SUBAPPLICATION InputOutputTesterButton_PWM_OPC_UA (* PWM Tester (OPC-UA): 8 unveraenderte digitale Eingaenge + 12 PWM-Ausgaenge (VT-Zahlenfeld/Balken/6 Ramp-Tasten je Kanal) *)
  (* Standard: 61499-2; Description: Copyright (c) 2026 Meisterschulen am Ostbahnhof This program and the accompanying materials are made available under the terms of the Eclipse Public License 2.0 which is available at https://www.eclipse.org/legal/epl-2.0/ SPDX-License-Identifier: EPL-2.0 *)
  (* Version 1.0, 2026-08-28, Franz Höpfinger, Meisterschulen am Ostbahnhof, initial API and implementation and/or initial documentation *)
  PACKAGE Meins::InputOutputTester::Button_PWM_OPC_UA;
  IMPORT Meins::InputOutputTester::Button_PWM_OPC_UA::SubStrings::I1_WRITE;
  IMPORT Meins::InputOutputTester::Button_PWM_OPC_UA::SubStrings::I2_WRITE;
  IMPORT Meins::InputOutputTester::Button_PWM_OPC_UA::SubStrings::I3_WRITE;
  IMPORT Meins::InputOutputTester::Button_PWM_OPC_UA::SubStrings::I4_WRITE;
  IMPORT Meins::InputOutputTester::Button_PWM_OPC_UA::SubStrings::I5_WRITE;
  IMPORT Meins::InputOutputTester::Button_PWM_OPC_UA::SubStrings::I6_WRITE;
  IMPORT Meins::InputOutputTester::Button_PWM_OPC_UA::SubStrings::I7_WRITE;
  IMPORT Meins::InputOutputTester::Button_PWM_OPC_UA::SubStrings::I8_WRITE;
  IMPORT Meins::InputOutputTester::Button_PWM_OPC_UA::SubStrings::PWM_Q01_READ;
  IMPORT Meins::InputOutputTester::Button_PWM_OPC_UA::SubStrings::PWM_Q01_WRITE;
  IMPORT Meins::InputOutputTester::Button_PWM_OPC_UA::SubStrings::PWM_Q01_SWITCH_READ;
  IMPORT Meins::InputOutputTester::Button_PWM_OPC_UA::SubStrings::PWM_Q01_SWITCH_WRITE;
  IMPORT Meins::InputOutputTester::Button_PWM_OPC_UA::SubStrings::PWM_Q01_STATUS_WRITE;
  IMPORT Meins::InputOutputTester::Button_PWM_OPC_UA::SubStrings::PWM_Q02_READ;
  IMPORT Meins::InputOutputTester::Button_PWM_OPC_UA::SubStrings::PWM_Q02_WRITE;
  IMPORT Meins::InputOutputTester::Button_PWM_OPC_UA::SubStrings::PWM_Q02_SWITCH_READ;
  IMPORT Meins::InputOutputTester::Button_PWM_OPC_UA::SubStrings::PWM_Q02_SWITCH_WRITE;
  IMPORT Meins::InputOutputTester::Button_PWM_OPC_UA::SubStrings::PWM_Q02_STATUS_WRITE;
  IMPORT Meins::InputOutputTester::Button_PWM_OPC_UA::SubStrings::PWM_Q03_READ;
  IMPORT Meins::InputOutputTester::Button_PWM_OPC_UA::SubStrings::PWM_Q03_WRITE;
  IMPORT Meins::InputOutputTester::Button_PWM_OPC_UA::SubStrings::PWM_Q03_SWITCH_READ;
  IMPORT Meins::InputOutputTester::Button_PWM_OPC_UA::SubStrings::PWM_Q03_SWITCH_WRITE;
  IMPORT Meins::InputOutputTester::Button_PWM_OPC_UA::SubStrings::PWM_Q03_STATUS_WRITE;
  IMPORT Meins::InputOutputTester::Button_PWM_OPC_UA::SubStrings::PWM_Q04_READ;
  IMPORT Meins::InputOutputTester::Button_PWM_OPC_UA::SubStrings::PWM_Q04_WRITE;
  IMPORT Meins::InputOutputTester::Button_PWM_OPC_UA::SubStrings::PWM_Q04_SWITCH_READ;
  IMPORT Meins::InputOutputTester::Button_PWM_OPC_UA::SubStrings::PWM_Q04_SWITCH_WRITE;
  IMPORT Meins::InputOutputTester::Button_PWM_OPC_UA::SubStrings::PWM_Q04_STATUS_WRITE;
  IMPORT Meins::InputOutputTester::Button_PWM_OPC_UA::SubStrings::PWM_Q05_READ;
  IMPORT Meins::InputOutputTester::Button_PWM_OPC_UA::SubStrings::PWM_Q05_WRITE;
  IMPORT Meins::InputOutputTester::Button_PWM_OPC_UA::SubStrings::PWM_Q05_SWITCH_READ;
  IMPORT Meins::InputOutputTester::Button_PWM_OPC_UA::SubStrings::PWM_Q05_SWITCH_WRITE;
  IMPORT Meins::InputOutputTester::Button_PWM_OPC_UA::SubStrings::PWM_Q05_STATUS_WRITE;
  IMPORT Meins::InputOutputTester::Button_PWM_OPC_UA::SubStrings::PWM_Q06_READ;
  IMPORT Meins::InputOutputTester::Button_PWM_OPC_UA::SubStrings::PWM_Q06_WRITE;
  IMPORT Meins::InputOutputTester::Button_PWM_OPC_UA::SubStrings::PWM_Q06_SWITCH_READ;
  IMPORT Meins::InputOutputTester::Button_PWM_OPC_UA::SubStrings::PWM_Q06_SWITCH_WRITE;
  IMPORT Meins::InputOutputTester::Button_PWM_OPC_UA::SubStrings::PWM_Q06_STATUS_WRITE;
  IMPORT Meins::InputOutputTester::Button_PWM_OPC_UA::SubStrings::PWM_Q07_READ;
  IMPORT Meins::InputOutputTester::Button_PWM_OPC_UA::SubStrings::PWM_Q07_WRITE;
  IMPORT Meins::InputOutputTester::Button_PWM_OPC_UA::SubStrings::PWM_Q07_SWITCH_READ;
  IMPORT Meins::InputOutputTester::Button_PWM_OPC_UA::SubStrings::PWM_Q07_SWITCH_WRITE;
  IMPORT Meins::InputOutputTester::Button_PWM_OPC_UA::SubStrings::PWM_Q07_STATUS_WRITE;
  IMPORT Meins::InputOutputTester::Button_PWM_OPC_UA::SubStrings::PWM_Q08_READ;
  IMPORT Meins::InputOutputTester::Button_PWM_OPC_UA::SubStrings::PWM_Q08_WRITE;
  IMPORT Meins::InputOutputTester::Button_PWM_OPC_UA::SubStrings::PWM_Q08_SWITCH_READ;
  IMPORT Meins::InputOutputTester::Button_PWM_OPC_UA::SubStrings::PWM_Q08_SWITCH_WRITE;
  IMPORT Meins::InputOutputTester::Button_PWM_OPC_UA::SubStrings::PWM_Q08_STATUS_WRITE;
  IMPORT Meins::InputOutputTester::Button_PWM_OPC_UA::SubStrings::PWM_Q09_READ;
  IMPORT Meins::InputOutputTester::Button_PWM_OPC_UA::SubStrings::PWM_Q09_WRITE;
  IMPORT Meins::InputOutputTester::Button_PWM_OPC_UA::SubStrings::PWM_Q09_SWITCH_READ;
  IMPORT Meins::InputOutputTester::Button_PWM_OPC_UA::SubStrings::PWM_Q09_SWITCH_WRITE;
  IMPORT Meins::InputOutputTester::Button_PWM_OPC_UA::SubStrings::PWM_Q09_STATUS_WRITE;
  IMPORT Meins::InputOutputTester::Button_PWM_OPC_UA::SubStrings::PWM_Q10_READ;
  IMPORT Meins::InputOutputTester::Button_PWM_OPC_UA::SubStrings::PWM_Q10_WRITE;
  IMPORT Meins::InputOutputTester::Button_PWM_OPC_UA::SubStrings::PWM_Q10_SWITCH_READ;
  IMPORT Meins::InputOutputTester::Button_PWM_OPC_UA::SubStrings::PWM_Q10_SWITCH_WRITE;
  IMPORT Meins::InputOutputTester::Button_PWM_OPC_UA::SubStrings::PWM_Q10_STATUS_WRITE;
  IMPORT Meins::InputOutputTester::Button_PWM_OPC_UA::SubStrings::PWM_Q11_READ;
  IMPORT Meins::InputOutputTester::Button_PWM_OPC_UA::SubStrings::PWM_Q11_WRITE;
  IMPORT Meins::InputOutputTester::Button_PWM_OPC_UA::SubStrings::PWM_Q11_SWITCH_READ;
  IMPORT Meins::InputOutputTester::Button_PWM_OPC_UA::SubStrings::PWM_Q11_SWITCH_WRITE;
  IMPORT Meins::InputOutputTester::Button_PWM_OPC_UA::SubStrings::PWM_Q11_STATUS_WRITE;
  IMPORT Meins::InputOutputTester::Button_PWM_OPC_UA::SubStrings::PWM_Q12_READ;
  IMPORT Meins::InputOutputTester::Button_PWM_OPC_UA::SubStrings::PWM_Q12_WRITE;
  IMPORT Meins::InputOutputTester::Button_PWM_OPC_UA::SubStrings::PWM_Q12_SWITCH_READ;
  IMPORT Meins::InputOutputTester::Button_PWM_OPC_UA::SubStrings::PWM_Q12_SWITCH_WRITE;
  IMPORT Meins::InputOutputTester::Button_PWM_OPC_UA::SubStrings::PWM_Q12_STATUS_WRITE;
  IMPORT Meins::InputOutputTester::Button_PWM_OPC_UA::SubStrings::Tick_WRITE;
  IMPORT Uebungen::const::UT::PWM12::DefaultPool_PWM12::Button_I01;
  IMPORT Uebungen::const::UT::PWM12::DefaultPool_PWM12::Button_I02;
  IMPORT Uebungen::const::UT::PWM12::DefaultPool_PWM12::Button_I03;
  IMPORT Uebungen::const::UT::PWM12::DefaultPool_PWM12::Button_I04;
  IMPORT Uebungen::const::UT::PWM12::DefaultPool_PWM12::Button_I05;
  IMPORT Uebungen::const::UT::PWM12::DefaultPool_PWM12::Button_I06;
  IMPORT Uebungen::const::UT::PWM12::DefaultPool_PWM12::Button_I07;
  IMPORT Uebungen::const::UT::PWM12::DefaultPool_PWM12::Button_I08;
  IMPORT Uebungen::const::UT::PWM12::DefaultPool_PWM12::NumberVariable_PWM_Q01;
  IMPORT Uebungen::const::UT::PWM12::DefaultPool_PWM12::Button_PWM_Q01_ZERO;
  IMPORT Uebungen::const::UT::PWM12::DefaultPool_PWM12::Button_PWM_Q01_DOWN_FAST;
  IMPORT Uebungen::const::UT::PWM12::DefaultPool_PWM12::Button_PWM_Q01_DOWN_SLOW;
  IMPORT Uebungen::const::UT::PWM12::DefaultPool_PWM12::Button_PWM_Q01_UP_SLOW;
  IMPORT Uebungen::const::UT::PWM12::DefaultPool_PWM12::Button_PWM_Q01_UP_FAST;
  IMPORT Uebungen::const::UT::PWM12::DefaultPool_PWM12::Button_PWM_Q01_FULL;
  IMPORT Uebungen::const::UT::PWM12::DefaultPool_PWM12::Button_PWM_Q01_SWITCH;
  IMPORT Uebungen::const::UT::PWM12::DefaultPool_PWM12::Button_PWM_Q01_STATUS;
  IMPORT Uebungen::const::UT::PWM12::DefaultPool_PWM12::NumberVariable_PWM_Q02;
  IMPORT Uebungen::const::UT::PWM12::DefaultPool_PWM12::Button_PWM_Q02_ZERO;
  IMPORT Uebungen::const::UT::PWM12::DefaultPool_PWM12::Button_PWM_Q02_DOWN_FAST;
  IMPORT Uebungen::const::UT::PWM12::DefaultPool_PWM12::Button_PWM_Q02_DOWN_SLOW;
  IMPORT Uebungen::const::UT::PWM12::DefaultPool_PWM12::Button_PWM_Q02_UP_SLOW;
  IMPORT Uebungen::const::UT::PWM12::DefaultPool_PWM12::Button_PWM_Q02_UP_FAST;
  IMPORT Uebungen::const::UT::PWM12::DefaultPool_PWM12::Button_PWM_Q02_FULL;
  IMPORT Uebungen::const::UT::PWM12::DefaultPool_PWM12::Button_PWM_Q02_SWITCH;
  IMPORT Uebungen::const::UT::PWM12::DefaultPool_PWM12::Button_PWM_Q02_STATUS;
  IMPORT Uebungen::const::UT::PWM12::DefaultPool_PWM12::NumberVariable_PWM_Q03;
  IMPORT Uebungen::const::UT::PWM12::DefaultPool_PWM12::Button_PWM_Q03_ZERO;
  IMPORT Uebungen::const::UT::PWM12::DefaultPool_PWM12::Button_PWM_Q03_DOWN_FAST;
  IMPORT Uebungen::const::UT::PWM12::DefaultPool_PWM12::Button_PWM_Q03_DOWN_SLOW;
  IMPORT Uebungen::const::UT::PWM12::DefaultPool_PWM12::Button_PWM_Q03_UP_SLOW;
  IMPORT Uebungen::const::UT::PWM12::DefaultPool_PWM12::Button_PWM_Q03_UP_FAST;
  IMPORT Uebungen::const::UT::PWM12::DefaultPool_PWM12::Button_PWM_Q03_FULL;
  IMPORT Uebungen::const::UT::PWM12::DefaultPool_PWM12::Button_PWM_Q03_SWITCH;
  IMPORT Uebungen::const::UT::PWM12::DefaultPool_PWM12::Button_PWM_Q03_STATUS;
  IMPORT Uebungen::const::UT::PWM12::DefaultPool_PWM12::NumberVariable_PWM_Q04;
  IMPORT Uebungen::const::UT::PWM12::DefaultPool_PWM12::Button_PWM_Q04_ZERO;
  IMPORT Uebungen::const::UT::PWM12::DefaultPool_PWM12::Button_PWM_Q04_DOWN_FAST;
  IMPORT Uebungen::const::UT::PWM12::DefaultPool_PWM12::Button_PWM_Q04_DOWN_SLOW;
  IMPORT Uebungen::const::UT::PWM12::DefaultPool_PWM12::Button_PWM_Q04_UP_SLOW;
  IMPORT Uebungen::const::UT::PWM12::DefaultPool_PWM12::Button_PWM_Q04_UP_FAST;
  IMPORT Uebungen::const::UT::PWM12::DefaultPool_PWM12::Button_PWM_Q04_FULL;
  IMPORT Uebungen::const::UT::PWM12::DefaultPool_PWM12::Button_PWM_Q04_SWITCH;
  IMPORT Uebungen::const::UT::PWM12::DefaultPool_PWM12::Button_PWM_Q04_STATUS;
  IMPORT Uebungen::const::UT::PWM12::DefaultPool_PWM12::NumberVariable_PWM_Q05;
  IMPORT Uebungen::const::UT::PWM12::DefaultPool_PWM12::Button_PWM_Q05_ZERO;
  IMPORT Uebungen::const::UT::PWM12::DefaultPool_PWM12::Button_PWM_Q05_DOWN_FAST;
  IMPORT Uebungen::const::UT::PWM12::DefaultPool_PWM12::Button_PWM_Q05_DOWN_SLOW;
  IMPORT Uebungen::const::UT::PWM12::DefaultPool_PWM12::Button_PWM_Q05_UP_SLOW;
  IMPORT Uebungen::const::UT::PWM12::DefaultPool_PWM12::Button_PWM_Q05_UP_FAST;
  IMPORT Uebungen::const::UT::PWM12::DefaultPool_PWM12::Button_PWM_Q05_FULL;
  IMPORT Uebungen::const::UT::PWM12::DefaultPool_PWM12::Button_PWM_Q05_SWITCH;
  IMPORT Uebungen::const::UT::PWM12::DefaultPool_PWM12::Button_PWM_Q05_STATUS;
  IMPORT Uebungen::const::UT::PWM12::DefaultPool_PWM12::NumberVariable_PWM_Q06;
  IMPORT Uebungen::const::UT::PWM12::DefaultPool_PWM12::Button_PWM_Q06_ZERO;
  IMPORT Uebungen::const::UT::PWM12::DefaultPool_PWM12::Button_PWM_Q06_DOWN_FAST;
  IMPORT Uebungen::const::UT::PWM12::DefaultPool_PWM12::Button_PWM_Q06_DOWN_SLOW;
  IMPORT Uebungen::const::UT::PWM12::DefaultPool_PWM12::Button_PWM_Q06_UP_SLOW;
  IMPORT Uebungen::const::UT::PWM12::DefaultPool_PWM12::Button_PWM_Q06_UP_FAST;
  IMPORT Uebungen::const::UT::PWM12::DefaultPool_PWM12::Button_PWM_Q06_FULL;
  IMPORT Uebungen::const::UT::PWM12::DefaultPool_PWM12::Button_PWM_Q06_SWITCH;
  IMPORT Uebungen::const::UT::PWM12::DefaultPool_PWM12::Button_PWM_Q06_STATUS;
  IMPORT Uebungen::const::UT::PWM12::DefaultPool_PWM12::NumberVariable_PWM_Q07;
  IMPORT Uebungen::const::UT::PWM12::DefaultPool_PWM12::Button_PWM_Q07_ZERO;
  IMPORT Uebungen::const::UT::PWM12::DefaultPool_PWM12::Button_PWM_Q07_DOWN_FAST;
  IMPORT Uebungen::const::UT::PWM12::DefaultPool_PWM12::Button_PWM_Q07_DOWN_SLOW;
  IMPORT Uebungen::const::UT::PWM12::DefaultPool_PWM12::Button_PWM_Q07_UP_SLOW;
  IMPORT Uebungen::const::UT::PWM12::DefaultPool_PWM12::Button_PWM_Q07_UP_FAST;
  IMPORT Uebungen::const::UT::PWM12::DefaultPool_PWM12::Button_PWM_Q07_FULL;
  IMPORT Uebungen::const::UT::PWM12::DefaultPool_PWM12::Button_PWM_Q07_SWITCH;
  IMPORT Uebungen::const::UT::PWM12::DefaultPool_PWM12::Button_PWM_Q07_STATUS;
  IMPORT Uebungen::const::UT::PWM12::DefaultPool_PWM12::NumberVariable_PWM_Q08;
  IMPORT Uebungen::const::UT::PWM12::DefaultPool_PWM12::Button_PWM_Q08_ZERO;
  IMPORT Uebungen::const::UT::PWM12::DefaultPool_PWM12::Button_PWM_Q08_DOWN_FAST;
  IMPORT Uebungen::const::UT::PWM12::DefaultPool_PWM12::Button_PWM_Q08_DOWN_SLOW;
  IMPORT Uebungen::const::UT::PWM12::DefaultPool_PWM12::Button_PWM_Q08_UP_SLOW;
  IMPORT Uebungen::const::UT::PWM12::DefaultPool_PWM12::Button_PWM_Q08_UP_FAST;
  IMPORT Uebungen::const::UT::PWM12::DefaultPool_PWM12::Button_PWM_Q08_FULL;
  IMPORT Uebungen::const::UT::PWM12::DefaultPool_PWM12::Button_PWM_Q08_SWITCH;
  IMPORT Uebungen::const::UT::PWM12::DefaultPool_PWM12::Button_PWM_Q08_STATUS;
  IMPORT Uebungen::const::UT::PWM12::DefaultPool_PWM12::NumberVariable_PWM_Q09;
  IMPORT Uebungen::const::UT::PWM12::DefaultPool_PWM12::Button_PWM_Q09_ZERO;
  IMPORT Uebungen::const::UT::PWM12::DefaultPool_PWM12::Button_PWM_Q09_DOWN_FAST;
  IMPORT Uebungen::const::UT::PWM12::DefaultPool_PWM12::Button_PWM_Q09_DOWN_SLOW;
  IMPORT Uebungen::const::UT::PWM12::DefaultPool_PWM12::Button_PWM_Q09_UP_SLOW;
  IMPORT Uebungen::const::UT::PWM12::DefaultPool_PWM12::Button_PWM_Q09_UP_FAST;
  IMPORT Uebungen::const::UT::PWM12::DefaultPool_PWM12::Button_PWM_Q09_FULL;
  IMPORT Uebungen::const::UT::PWM12::DefaultPool_PWM12::Button_PWM_Q09_SWITCH;
  IMPORT Uebungen::const::UT::PWM12::DefaultPool_PWM12::Button_PWM_Q09_STATUS;
  IMPORT Uebungen::const::UT::PWM12::DefaultPool_PWM12::NumberVariable_PWM_Q10;
  IMPORT Uebungen::const::UT::PWM12::DefaultPool_PWM12::Button_PWM_Q10_ZERO;
  IMPORT Uebungen::const::UT::PWM12::DefaultPool_PWM12::Button_PWM_Q10_DOWN_FAST;
  IMPORT Uebungen::const::UT::PWM12::DefaultPool_PWM12::Button_PWM_Q10_DOWN_SLOW;
  IMPORT Uebungen::const::UT::PWM12::DefaultPool_PWM12::Button_PWM_Q10_UP_SLOW;
  IMPORT Uebungen::const::UT::PWM12::DefaultPool_PWM12::Button_PWM_Q10_UP_FAST;
  IMPORT Uebungen::const::UT::PWM12::DefaultPool_PWM12::Button_PWM_Q10_FULL;
  IMPORT Uebungen::const::UT::PWM12::DefaultPool_PWM12::Button_PWM_Q10_SWITCH;
  IMPORT Uebungen::const::UT::PWM12::DefaultPool_PWM12::Button_PWM_Q10_STATUS;
  IMPORT Uebungen::const::UT::PWM12::DefaultPool_PWM12::NumberVariable_PWM_Q11;
  IMPORT Uebungen::const::UT::PWM12::DefaultPool_PWM12::Button_PWM_Q11_ZERO;
  IMPORT Uebungen::const::UT::PWM12::DefaultPool_PWM12::Button_PWM_Q11_DOWN_FAST;
  IMPORT Uebungen::const::UT::PWM12::DefaultPool_PWM12::Button_PWM_Q11_DOWN_SLOW;
  IMPORT Uebungen::const::UT::PWM12::DefaultPool_PWM12::Button_PWM_Q11_UP_SLOW;
  IMPORT Uebungen::const::UT::PWM12::DefaultPool_PWM12::Button_PWM_Q11_UP_FAST;
  IMPORT Uebungen::const::UT::PWM12::DefaultPool_PWM12::Button_PWM_Q11_FULL;
  IMPORT Uebungen::const::UT::PWM12::DefaultPool_PWM12::Button_PWM_Q11_SWITCH;
  IMPORT Uebungen::const::UT::PWM12::DefaultPool_PWM12::Button_PWM_Q11_STATUS;
  IMPORT Uebungen::const::UT::PWM12::DefaultPool_PWM12::NumberVariable_PWM_Q12;
  IMPORT Uebungen::const::UT::PWM12::DefaultPool_PWM12::Button_PWM_Q12_ZERO;
  IMPORT Uebungen::const::UT::PWM12::DefaultPool_PWM12::Button_PWM_Q12_DOWN_FAST;
  IMPORT Uebungen::const::UT::PWM12::DefaultPool_PWM12::Button_PWM_Q12_DOWN_SLOW;
  IMPORT Uebungen::const::UT::PWM12::DefaultPool_PWM12::Button_PWM_Q12_UP_SLOW;
  IMPORT Uebungen::const::UT::PWM12::DefaultPool_PWM12::Button_PWM_Q12_UP_FAST;
  IMPORT Uebungen::const::UT::PWM12::DefaultPool_PWM12::Button_PWM_Q12_FULL;
  IMPORT Uebungen::const::UT::PWM12::DefaultPool_PWM12::Button_PWM_Q12_SWITCH;
  IMPORT Uebungen::const::UT::PWM12::DefaultPool_PWM12::Button_PWM_Q12_STATUS;
  IMPORT Uebungen::const::UT::PWM12::DefaultPool_PWM12::OutputNumber_Tick;
  IMPORT logiBUS::io::DI::logiBUS_DI::Input_I1;
  IMPORT logiBUS::io::DI::logiBUS_DI::Input_I2;
  IMPORT logiBUS::io::DI::logiBUS_DI::Input_I3;
  IMPORT logiBUS::io::DI::logiBUS_DI::Input_I4;
  IMPORT logiBUS::io::DI::logiBUS_DI::Input_I5;
  IMPORT logiBUS::io::DI::logiBUS_DI::Input_I6;
  IMPORT logiBUS::io::DI::logiBUS_DI::Input_I7;
  IMPORT logiBUS::io::DI::logiBUS_DI::Input_I8;
  IMPORT logiBUS::io::DQ::logiBUS_DO::Output_Q1;
  IMPORT logiBUS::io::DQ::logiBUS_DO::Output_Q2;
  IMPORT logiBUS::io::DQ::logiBUS_DO::Output_Q3;
  IMPORT logiBUS::io::DQ::logiBUS_DO::Output_Q4;
  IMPORT logiBUS::io::DQ::logiBUS_DO::Output_Q5;
  IMPORT logiBUS::io::DQ::logiBUS_DO::Output_Q6;
  IMPORT logiBUS::io::DQ::logiBUS_DO::Output_Q7;
  IMPORT logiBUS::io::DQ::logiBUS_DO::Output_Q8;
  IMPORT logiBUS::io::DQ::logiBUS_DO::Output_Q9;
  IMPORT logiBUS::io::DQ::logiBUS_DO::Output_Q10;
  IMPORT logiBUS::io::DQ::logiBUS_DO::Output_Q11;
  IMPORT logiBUS::io::DQ::logiBUS_DO::Output_Q12;
  SUBAPPS
    Input_I1 : MyLib::sys::logiBUS_IXA_BG_OPC(u16ObjId := Button_I01, Input := Input_I1, ID_WRITE := I1_WRITE);
    Input_I2 : MyLib::sys::logiBUS_IXA_BG_OPC(u16ObjId := Button_I02, Input := Input_I2, ID_WRITE := I2_WRITE);
    Input_I3 : MyLib::sys::logiBUS_IXA_BG_OPC(u16ObjId := Button_I03, Input := Input_I3, ID_WRITE := I3_WRITE);
    Input_I4 : MyLib::sys::logiBUS_IXA_BG_OPC(u16ObjId := Button_I04, Input := Input_I4, ID_WRITE := I4_WRITE);
    Input_I5 : MyLib::sys::logiBUS_IXA_BG_OPC(u16ObjId := Button_I05, Input := Input_I5, ID_WRITE := I5_WRITE);
    Input_I6 : MyLib::sys::logiBUS_IXA_BG_OPC(u16ObjId := Button_I06, Input := Input_I6, ID_WRITE := I6_WRITE);
    Input_I7 : MyLib::sys::logiBUS_IXA_BG_OPC(u16ObjId := Button_I07, Input := Input_I7, ID_WRITE := I7_WRITE);
    Input_I8 : MyLib::sys::logiBUS_IXA_BG_OPC(u16ObjId := Button_I08, Input := Input_I8, ID_WRITE := I8_WRITE);
    Output_Q1 : MyLib::sys::RampLimitFS_TO_logiBUS_QDA_PWM_OPC(u16ObjId_VALUEVAR := NumberVariable_PWM_Q01, u16ObjId_SWITCH := Button_PWM_Q01_SWITCH, u16ObjId_STATUS := Button_PWM_Q01_STATUS, bDefaultEnabled := TRUE, u16ObjId_ZERO := Button_PWM_Q01_ZERO, u16ObjId_DOWN_FAST := Button_PWM_Q01_DOWN_FAST, u16ObjId_DOWN_SLOW := Button_PWM_Q01_DOWN_SLOW, u16ObjId_UP_SLOW := Button_PWM_Q01_UP_SLOW, u16ObjId_UP_FAST := Button_PWM_Q01_UP_FAST, u16ObjId_FULL := Button_PWM_Q01_FULL, Output := Output_Q1, ID_READ := PWM_Q01_READ, ID_WRITE := PWM_Q01_WRITE, ID_SWITCH_READ := PWM_Q01_SWITCH_READ, ID_SWITCH_WRITE := PWM_Q01_SWITCH_WRITE, ID_STATUS_WRITE := PWM_Q01_STATUS_WRITE);
    Output_Q2 : MyLib::sys::RampLimitFS_TO_logiBUS_QDA_PWM_OPC(u16ObjId_VALUEVAR := NumberVariable_PWM_Q02, u16ObjId_SWITCH := Button_PWM_Q02_SWITCH, u16ObjId_STATUS := Button_PWM_Q02_STATUS, bDefaultEnabled := TRUE, u16ObjId_ZERO := Button_PWM_Q02_ZERO, u16ObjId_DOWN_FAST := Button_PWM_Q02_DOWN_FAST, u16ObjId_DOWN_SLOW := Button_PWM_Q02_DOWN_SLOW, u16ObjId_UP_SLOW := Button_PWM_Q02_UP_SLOW, u16ObjId_UP_FAST := Button_PWM_Q02_UP_FAST, u16ObjId_FULL := Button_PWM_Q02_FULL, Output := Output_Q2, ID_READ := PWM_Q02_READ, ID_WRITE := PWM_Q02_WRITE, ID_SWITCH_READ := PWM_Q02_SWITCH_READ, ID_SWITCH_WRITE := PWM_Q02_SWITCH_WRITE, ID_STATUS_WRITE := PWM_Q02_STATUS_WRITE);
    Output_Q3 : MyLib::sys::RampLimitFS_TO_logiBUS_QDA_PWM_OPC(u16ObjId_VALUEVAR := NumberVariable_PWM_Q03, u16ObjId_SWITCH := Button_PWM_Q03_SWITCH, u16ObjId_STATUS := Button_PWM_Q03_STATUS, bDefaultEnabled := TRUE, u16ObjId_ZERO := Button_PWM_Q03_ZERO, u16ObjId_DOWN_FAST := Button_PWM_Q03_DOWN_FAST, u16ObjId_DOWN_SLOW := Button_PWM_Q03_DOWN_SLOW, u16ObjId_UP_SLOW := Button_PWM_Q03_UP_SLOW, u16ObjId_UP_FAST := Button_PWM_Q03_UP_FAST, u16ObjId_FULL := Button_PWM_Q03_FULL, Output := Output_Q3, ID_READ := PWM_Q03_READ, ID_WRITE := PWM_Q03_WRITE, ID_SWITCH_READ := PWM_Q03_SWITCH_READ, ID_SWITCH_WRITE := PWM_Q03_SWITCH_WRITE, ID_STATUS_WRITE := PWM_Q03_STATUS_WRITE);
    Output_Q4 : MyLib::sys::RampLimitFS_TO_logiBUS_QDA_PWM_OPC(u16ObjId_VALUEVAR := NumberVariable_PWM_Q04, u16ObjId_SWITCH := Button_PWM_Q04_SWITCH, u16ObjId_STATUS := Button_PWM_Q04_STATUS, bDefaultEnabled := TRUE, u16ObjId_ZERO := Button_PWM_Q04_ZERO, u16ObjId_DOWN_FAST := Button_PWM_Q04_DOWN_FAST, u16ObjId_DOWN_SLOW := Button_PWM_Q04_DOWN_SLOW, u16ObjId_UP_SLOW := Button_PWM_Q04_UP_SLOW, u16ObjId_UP_FAST := Button_PWM_Q04_UP_FAST, u16ObjId_FULL := Button_PWM_Q04_FULL, Output := Output_Q4, ID_READ := PWM_Q04_READ, ID_WRITE := PWM_Q04_WRITE, ID_SWITCH_READ := PWM_Q04_SWITCH_READ, ID_SWITCH_WRITE := PWM_Q04_SWITCH_WRITE, ID_STATUS_WRITE := PWM_Q04_STATUS_WRITE);
    Output_Q5 : MyLib::sys::RampLimitFS_TO_logiBUS_QDA_PWM_OPC(u16ObjId_VALUEVAR := NumberVariable_PWM_Q05, u16ObjId_SWITCH := Button_PWM_Q05_SWITCH, u16ObjId_STATUS := Button_PWM_Q05_STATUS, bDefaultEnabled := TRUE, u16ObjId_ZERO := Button_PWM_Q05_ZERO, u16ObjId_DOWN_FAST := Button_PWM_Q05_DOWN_FAST, u16ObjId_DOWN_SLOW := Button_PWM_Q05_DOWN_SLOW, u16ObjId_UP_SLOW := Button_PWM_Q05_UP_SLOW, u16ObjId_UP_FAST := Button_PWM_Q05_UP_FAST, u16ObjId_FULL := Button_PWM_Q05_FULL, Output := Output_Q5, ID_READ := PWM_Q05_READ, ID_WRITE := PWM_Q05_WRITE, ID_SWITCH_READ := PWM_Q05_SWITCH_READ, ID_SWITCH_WRITE := PWM_Q05_SWITCH_WRITE, ID_STATUS_WRITE := PWM_Q05_STATUS_WRITE);
    Output_Q6 : MyLib::sys::RampLimitFS_TO_logiBUS_QDA_PWM_OPC(u16ObjId_VALUEVAR := NumberVariable_PWM_Q06, u16ObjId_SWITCH := Button_PWM_Q06_SWITCH, u16ObjId_STATUS := Button_PWM_Q06_STATUS, bDefaultEnabled := TRUE, u16ObjId_ZERO := Button_PWM_Q06_ZERO, u16ObjId_DOWN_FAST := Button_PWM_Q06_DOWN_FAST, u16ObjId_DOWN_SLOW := Button_PWM_Q06_DOWN_SLOW, u16ObjId_UP_SLOW := Button_PWM_Q06_UP_SLOW, u16ObjId_UP_FAST := Button_PWM_Q06_UP_FAST, u16ObjId_FULL := Button_PWM_Q06_FULL, Output := Output_Q6, ID_READ := PWM_Q06_READ, ID_WRITE := PWM_Q06_WRITE, ID_SWITCH_READ := PWM_Q06_SWITCH_READ, ID_SWITCH_WRITE := PWM_Q06_SWITCH_WRITE, ID_STATUS_WRITE := PWM_Q06_STATUS_WRITE);
    Output_Q7 : MyLib::sys::RampLimitFS_TO_logiBUS_QDA_PWM_OPC(u16ObjId_VALUEVAR := NumberVariable_PWM_Q07, u16ObjId_SWITCH := Button_PWM_Q07_SWITCH, u16ObjId_STATUS := Button_PWM_Q07_STATUS, bDefaultEnabled := TRUE, u16ObjId_ZERO := Button_PWM_Q07_ZERO, u16ObjId_DOWN_FAST := Button_PWM_Q07_DOWN_FAST, u16ObjId_DOWN_SLOW := Button_PWM_Q07_DOWN_SLOW, u16ObjId_UP_SLOW := Button_PWM_Q07_UP_SLOW, u16ObjId_UP_FAST := Button_PWM_Q07_UP_FAST, u16ObjId_FULL := Button_PWM_Q07_FULL, Output := Output_Q7, ID_READ := PWM_Q07_READ, ID_WRITE := PWM_Q07_WRITE, ID_SWITCH_READ := PWM_Q07_SWITCH_READ, ID_SWITCH_WRITE := PWM_Q07_SWITCH_WRITE, ID_STATUS_WRITE := PWM_Q07_STATUS_WRITE);
    Output_Q8 : MyLib::sys::RampLimitFS_TO_logiBUS_QDA_PWM_OPC(u16ObjId_VALUEVAR := NumberVariable_PWM_Q08, u16ObjId_SWITCH := Button_PWM_Q08_SWITCH, u16ObjId_STATUS := Button_PWM_Q08_STATUS, bDefaultEnabled := TRUE, u16ObjId_ZERO := Button_PWM_Q08_ZERO, u16ObjId_DOWN_FAST := Button_PWM_Q08_DOWN_FAST, u16ObjId_DOWN_SLOW := Button_PWM_Q08_DOWN_SLOW, u16ObjId_UP_SLOW := Button_PWM_Q08_UP_SLOW, u16ObjId_UP_FAST := Button_PWM_Q08_UP_FAST, u16ObjId_FULL := Button_PWM_Q08_FULL, Output := Output_Q8, ID_READ := PWM_Q08_READ, ID_WRITE := PWM_Q08_WRITE, ID_SWITCH_READ := PWM_Q08_SWITCH_READ, ID_SWITCH_WRITE := PWM_Q08_SWITCH_WRITE, ID_STATUS_WRITE := PWM_Q08_STATUS_WRITE);
    Output_Q9 : MyLib::sys::RampLimitFS_TO_logiBUS_QDA_PWM_OPC(u16ObjId_VALUEVAR := NumberVariable_PWM_Q09, u16ObjId_SWITCH := Button_PWM_Q09_SWITCH, u16ObjId_STATUS := Button_PWM_Q09_STATUS, bDefaultEnabled := FALSE, u16ObjId_ZERO := Button_PWM_Q09_ZERO, u16ObjId_DOWN_FAST := Button_PWM_Q09_DOWN_FAST, u16ObjId_DOWN_SLOW := Button_PWM_Q09_DOWN_SLOW, u16ObjId_UP_SLOW := Button_PWM_Q09_UP_SLOW, u16ObjId_UP_FAST := Button_PWM_Q09_UP_FAST, u16ObjId_FULL := Button_PWM_Q09_FULL, Output := Output_Q9, ID_READ := PWM_Q09_READ, ID_WRITE := PWM_Q09_WRITE, ID_SWITCH_READ := PWM_Q09_SWITCH_READ, ID_SWITCH_WRITE := PWM_Q09_SWITCH_WRITE, ID_STATUS_WRITE := PWM_Q09_STATUS_WRITE);
    Output_Q10 : MyLib::sys::RampLimitFS_TO_logiBUS_QDA_PWM_OPC(u16ObjId_VALUEVAR := NumberVariable_PWM_Q10, u16ObjId_SWITCH := Button_PWM_Q10_SWITCH, u16ObjId_STATUS := Button_PWM_Q10_STATUS, bDefaultEnabled := FALSE, u16ObjId_ZERO := Button_PWM_Q10_ZERO, u16ObjId_DOWN_FAST := Button_PWM_Q10_DOWN_FAST, u16ObjId_DOWN_SLOW := Button_PWM_Q10_DOWN_SLOW, u16ObjId_UP_SLOW := Button_PWM_Q10_UP_SLOW, u16ObjId_UP_FAST := Button_PWM_Q10_UP_FAST, u16ObjId_FULL := Button_PWM_Q10_FULL, Output := Output_Q10, ID_READ := PWM_Q10_READ, ID_WRITE := PWM_Q10_WRITE, ID_SWITCH_READ := PWM_Q10_SWITCH_READ, ID_SWITCH_WRITE := PWM_Q10_SWITCH_WRITE, ID_STATUS_WRITE := PWM_Q10_STATUS_WRITE);
    Output_Q11 : MyLib::sys::RampLimitFS_TO_logiBUS_QDA_PWM_OPC(u16ObjId_VALUEVAR := NumberVariable_PWM_Q11, u16ObjId_SWITCH := Button_PWM_Q11_SWITCH, u16ObjId_STATUS := Button_PWM_Q11_STATUS, bDefaultEnabled := FALSE, u16ObjId_ZERO := Button_PWM_Q11_ZERO, u16ObjId_DOWN_FAST := Button_PWM_Q11_DOWN_FAST, u16ObjId_DOWN_SLOW := Button_PWM_Q11_DOWN_SLOW, u16ObjId_UP_SLOW := Button_PWM_Q11_UP_SLOW, u16ObjId_UP_FAST := Button_PWM_Q11_UP_FAST, u16ObjId_FULL := Button_PWM_Q11_FULL, Output := Output_Q11, ID_READ := PWM_Q11_READ, ID_WRITE := PWM_Q11_WRITE, ID_SWITCH_READ := PWM_Q11_SWITCH_READ, ID_SWITCH_WRITE := PWM_Q11_SWITCH_WRITE, ID_STATUS_WRITE := PWM_Q11_STATUS_WRITE);
    Output_Q12 : MyLib::sys::RampLimitFS_TO_logiBUS_QDA_PWM_OPC(u16ObjId_VALUEVAR := NumberVariable_PWM_Q12, u16ObjId_SWITCH := Button_PWM_Q12_SWITCH, u16ObjId_STATUS := Button_PWM_Q12_STATUS, bDefaultEnabled := FALSE, u16ObjId_ZERO := Button_PWM_Q12_ZERO, u16ObjId_DOWN_FAST := Button_PWM_Q12_DOWN_FAST, u16ObjId_DOWN_SLOW := Button_PWM_Q12_DOWN_SLOW, u16ObjId_UP_SLOW := Button_PWM_Q12_UP_SLOW, u16ObjId_UP_FAST := Button_PWM_Q12_UP_FAST, u16ObjId_FULL := Button_PWM_Q12_FULL, Output := Output_Q12, ID_READ := PWM_Q12_READ, ID_WRITE := PWM_Q12_WRITE, ID_SWITCH_READ := PWM_Q12_SWITCH_READ, ID_SWITCH_WRITE := PWM_Q12_SWITCH_WRITE, ID_STATUS_WRITE := PWM_Q12_STATUS_WRITE);
    SystemTickSender : MyLib::sys::SystemTickSender_ISO_OPC(u16ObjId := OutputNumber_Tick, ID_WRITE := Tick_WRITE);
  END_SUBAPPS
END_SUBAPPLICATION
